RoboDK station: ur16e.rdk

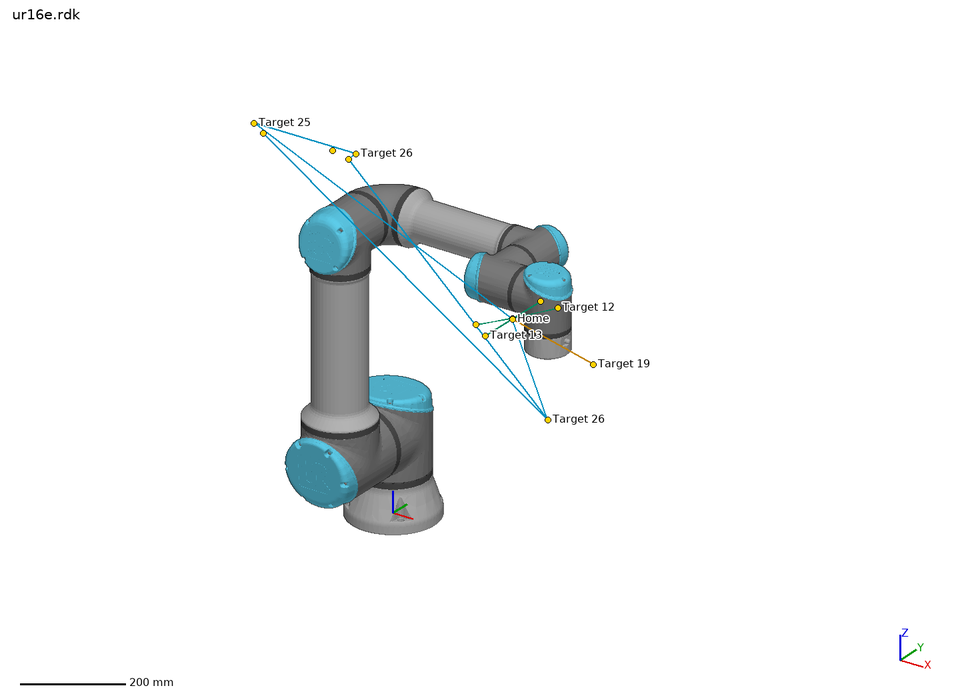
[picture v0: the station drawn from its stored meshes, robots at their saved joint values, targets as dots, program paths as lines]
Station ur16e (saved by RoboDK 5.9.4). Poses are relative to the parent item; angles as X-Y-Z fixed-axis rotations.
  - frame UR16e Base at (0, 0, 0) mm
    - robot UR16e: 6 axes, payload 16 kg, reach 900 mm, repeatability 0.05 mm, weight 33.1 kg
        modified DH rows (alpha deg, a mm, theta deg, d mm): 0, 0, 0, 180.7; 90, 0, 180, 0; 0, 478.4, 0, 0; 0, 360, 0, 174.15; -90, 0, 0, 119.85; 90, 0, 180, 116.55
        joint limits [-360, -360, -360, -360, -360, -360] to [360, 360, 360, 360, 360, 360]; home [0, -90, -90, 0, 90, 0]; saved at [0, -90, -90, -90, 90, 0]
      - tool TCP_FLANGE, TCP at (0, 0, 0) mm
      - tool TCP_GRIPKIT, TCP at (0, 0, 143) mm
    - target Home (joint target) at (479.85, -290.7, 659.1) mm, rotated rx 0 ry -90 rz 90 deg; joints [0, -90, -90, -90, 0, 0] of UR16e
    - frame W_sin at (0, 0, 0) mm
      - target Target 2 (joint target) at (479.81, -290.7, 659.22) mm, rotated rx -90 ry -89.95 rz 180 deg; joints [0, -90.07, -91.6, -83.25, 0, -5.03] of UR16e
      - target Target 3 (joint target) at (479.85, -290.7, 659.15) mm, rotated rx 90 ry -89.83 rz 0 deg; joints [0, -90.52, -93.9, -72.16, 0, -13.59] of UR16e
      - target Target 4 (joint target) at (479.81, -290.7, 659.16) mm, rotated rx -90 ry -89.72 rz 180 deg; joints [0, -91.9, -96.43, -55.7, 0, -25.69] of UR16e
      - target Target 5 (joint target) at (479.85, -290.7, 659.16) mm, rotated rx 90 ry -89.45 rz 0 deg; joints [0, -94.27, -97.79, -38.21, 0, -40.28] of UR16e
      - target Target 6 (joint target) at (479.8, -290.7, 659.2) mm, rotated rx 90 ry -89.55 rz 0 deg; joints [0, -96.9, -97.7, -23.5, 0, -52.35] of UR16e
      - target Target 7 (joint target) at (479.77, -290.7, 659.23) mm, rotated rx 90 ry -89.54 rz 0 deg; joints [0, -99.43, -96.64, -11.49, 0, -62.9] of UR16e
      - target Target 8 (joint target) at (479.85, -290.7, 659.15) mm, rotated rx 90 ry -89.97 rz 0 deg; joints [0, -102.33, -94.48, 0.79, 0, -74.01] of UR16e
      - target Target 9 (joint target) at (479.8, -290.7, 659.19) mm, rotated rx -90 ry -89.76 rz 180 deg; joints [0, -104.9, -91.74, 10.96, 0, -84.08] of UR16e
      - target Target 10 (joint target) at (479.82, -290.7, 659.16) mm, rotated rx -90 ry -89.48 rz 180 deg; joints [0, -106.17, -90.1, 15.79, 0, -89] of UR16e
    - frame W_lock at (0, 0, 0) mm
      - target Target 11 (Cartesian target) at (437.41, -351.22, 659.18) mm, rotated rx -90 ry -89.99 rz 172.45 deg; joints [-7.55, -89.99, -90, -90, 0, 0] of UR16e
      - target Target 12 (Cartesian target) at (523.2, -202.33, 659.18) mm, rotated rx -90 ry -89.99 rz -169.93 deg; joints [10.07, -89.99, -90, -90, 0, 0] of UR16e
      - target Target 13 (joint target) at (479.82, -379.57, 659.16) mm, rotated rx -90 ry -89.48 rz 180 deg; joints [-10.172, -110.79, -83.463, 14.254, 10.172, -89.48] of UR16e
      - target Target 14 (Cartesian target) at (479.82, -290.7, 659.16) mm, rotated rx -90 ry -89.48 rz 180 deg; joints [0, -106.17, -90.1, 15.79, 0, -89] of UR16e
    - target Target 15 (Cartesian target) at (479.82, -197.93, 659.16) mm, rotated rx -90 ry -89.48 rz 180 deg; joints [11.342, -103.374, -93.887, 17.26, -11.342, -89.48] of UR16e
    - target Target 16 (Cartesian target) at (479.85, -290.7, 659.1) mm, rotated rx 0 ry -90 rz 90 deg; joints [140.106, -71.743, 48.176, 23.567, 140.106, 90] of UR16e
    - target Target 17 (Cartesian target) at (479.85, -290.7, 659.1) mm, rotated rx 0 ry -90 rz 90 deg; joints [0, -149.208, 48.176, -258.968, 0, 90] of UR16e
    - target Target 18 (Cartesian target) at (479.85, -290.7, 659.1) mm, rotated rx 0 ry -90 rz 90 deg; joints [140.106, 0.173, -89.942, -90.231, -140.106, -90] of UR16e
    - target Target 19 (Cartesian target) at (718.72, -364.31, 659.23) mm, rotated rx -90 ry -89.99 rz 172.45 deg; joints [-5.737, -150.892, -8.627, -20.481, -1.813, -89.99] of UR16e
    - target Target 20 (Cartesian target) at (718.72, -364.31, 659.23) mm, rotated rx -90 ry -89.99 rz 172.45 deg; joints [-5.737, -158.299, 8.627, -30.329, -1.813, -89.99] of UR16e
    - target Target 25 (Cartesian target) at (-117.36, -291.5, 905.56) mm, rotated rx -89.53 ry -89.98 rz 179.99 deg; joints [0.388, -43.217, -86.375, -50.281, 0.073, -90.107] of UR16e
    - target Target 26 (Cartesian target) at (117.39, -289.61, 905.64) mm, rotated rx -89.53 ry -89.98 rz 179.99 deg; joints [0.536, -65.025, -86.539, -28.559, -0.076, -89.858] of UR16e
    - target Target 23 (Cartesian target) at (72.81, -304.63, 905.62) mm, rotated rx -89.53 ry -89.98 rz 179.99 deg; joints [-9.211, -63.604, -87.028, -29.367, 9.67, -89.981] of UR16e
    - target Target 24 (Cartesian target) at (118.23, -316.73, 905.64) mm, rotated rx -89.53 ry -89.98 rz 179.99 deg; joints [-10.99, -69.163, -84.808, -26.028, 11.45, -89.981] of UR16e
    - target Target 25 (Cartesian target) at (-77.53, -318.3, 905.57) mm, rotated rx -89.53 ry -89.98 rz 179.99 deg; joints [-57.693, -66.506, -85.985, -27.509, 58.153, -89.98] of UR16e
    - frame J_vs_L at (0, 0, 0) mm
      - target Target 26 (joint target) at (479.85, -174.15, 399.55) mm, rotated rx -180 ry 0 rz -90 deg; joints [0, -90, -90, -90, 90, 0] of UR16e
      - target Target 27 (Cartesian target) at (479.85, -174.15, 399.55) mm, rotated rx -180 ry 0 rz -90 deg; joints [0, -90, -90, -90, 90, 0] of UR16e
  - program J_vs_L (4 instructions, listed below)
  - program W_sin (21 instructions, listed below)
  - program W_lock (12 instructions, listed below)
  - program Conf (7 instructions, listed below)
  - program E_sin (11 instructions, listed below)
  - program S_sin (18 instructions, listed below)
  - program Home (2 instructions, listed below)
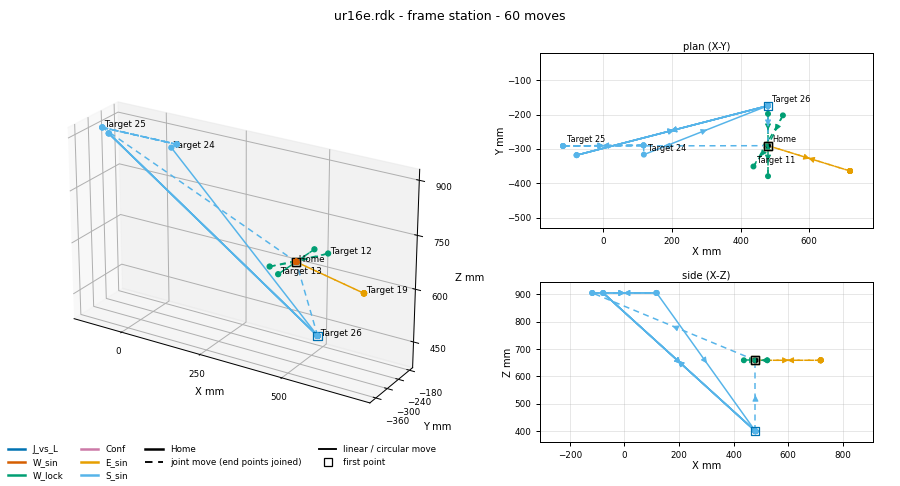
[picture p0: tool path of ur16e.rdk in frame station, 60 of 60 moves have a stored position in this frame; points joined in program order, loops and branches not executed]

--- program J_vs_L (robot UR16e) ---
  Set Ref.: J_vs_L
  Set Tool: TCP_GRIPKIT
  MoveJ (Target 26)
  MoveJ (Target 2) -> target Target 27

--- program W_sin (robot UR16e) ---
  Set Ref.: W_sin
  Set Tool: TCP_FLANGE
  MoveJ (Home)
  MoveJ (Target 2)
  MoveJ (Target 3)
  MoveJ (Target 4)
  MoveJ (Target 5)
  MoveJ (Target 6)
  MoveJ (Target 7)
  MoveJ (Target 8)
  MoveJ (Target 9)
  MoveJ (Target 10)
  MoveJ (Target 9)
  MoveJ (Target 8)
  MoveJ (Target 7)
  MoveJ (Target 6)
  MoveJ (Target 5)
  MoveJ (Target 4)
  MoveJ (Target 3)
  MoveJ (Target 2)
  MoveJ (Home)

--- program W_lock (robot UR16e) ---
  Set Ref.: W_lock
  Set Tool: TCP_FLANGE
  MoveJ (Target 1) -> target Home
  MoveJ (Target 11)
  MoveJ (Target 12)
  MoveJ (Target 1) -> target Home
  Pause 500 ms
  MoveJ (Target 10)
  MoveJ (Target 13)
  MoveJ (Target 15)
  MoveJ (Target 10)
  Pause 500 ms

--- program Conf (robot UR16e) ---
  Set Ref.: UR16e Base
  Set Tool: TCP_FLANGE
  MoveJ (Home)
  MoveJ (Target 16)
  MoveJ (Target 18)
  MoveJ (Target 17)
  MoveJ (Home)

--- program E_sin (robot UR16e) ---
  Set Ref.: UR16e Base
  Set Tool: TCP_FLANGE
  MoveJ (Home)
  MoveJ (Target 19)
  MoveJ (Target 20)
  MoveJ (Target 19)
  MoveJ (Target 20)
  MoveJ (Target 19)
  MoveJ (Target 20)
  MoveJ (Target 19)
  MoveJ (Home)

--- program S_sin (robot UR16e) ---
  Set Ref.: UR16e Base
  Set Tool: TCP_FLANGE
  MoveJ (Home)
  MoveJ (Target 25)
  MoveJ (Target 26)
  MoveJ (Target 25)
  MoveJ (Target 26)
  MoveJ (Target 25)
  MoveJ (Target 26)
  MoveJ (Target 24)
  MoveL (Target 26)
  MoveL (Target 25)
  MoveL (Target 26)
  MoveL (Target 25)
  MoveL (Target 26)
  MoveL (Target 25)
  MoveL (Target 26)
  MoveJ (Home)

--- program Home (robot UR16e) ---
  Set Ref.: UR16e Base
  MoveJ (Home)
